Staubli VAL3: recvData.pgx

public program recvData(sio& x_sTcpSocket (dimensions=1), num& x_nData[] (dimensions=1), num& x_nConnFlag (dimensions=1), bool& x_bValidFlag (dimensions=1))
  local num l_nByte
  local num l_nBytesRecv
  local num l_nIndex
begin
  // attempt to receive data on specified socket
  l_nBytesRecv=0
  l_nIndex=0
  x_bValidFlag=false

  while (l_nBytesRecv<size(x_nData))
    l_nIndex=sioGet(x_sTcpSocket,l_nByte)
    if (l_nIndex==1)
      x_nData[l_nBytesRecv]=l_nByte
      l_nBytesRecv=l_nBytesRecv+l_nIndex
      // received a byte, set flag to indicate connection
      x_nConnFlag=1
    elseIf (l_nIndex==-1)
      // error or timeout, indicate only if connection previously established
      if (x_nConnFlag==1)
        x_nConnFlag=-1
        // close connection properly (to avoid CLOSE_WAIT)
        clearBuffer(x_sTcpSocket)
      endIf
      return
    elseIf (l_nIndex>1)
      popUpMsg("sioGet() returned > 1")
      //else
      //  popUpMsg("sioGet() returned 0")
    endIf
  endWhile
  x_bValidFlag=true
end
